{attribute 'GeneratedUsingTerminal: EP5001-0002-0016'}
{attribute addProperty BoxType "EP5001-0002-0016"}
{attribute addProperty Id "SSI_InputsAT %I*SSI_Inputs_0E3D8E3310WcStateAT %I*WcState_9091E0EB2InfoDataAT %I*InfoData_32EB74EA10"}
{attribute addProperty CRC "187224199"}
{attribute addProperty Size "22"}
TYPE EP5001_0B28D087 EXTENDS EtcSlaveTerminalBase_947E5A46 :
STRUCT
	{attribute addProperty Name "SSI_Inputs"}
	SSI_Inputs : SSI_Inputs_0E3D8E33;
	{attribute addProperty Name "WcState"}
	WcState : WcState_9091E0EB;
	{attribute addProperty Name "InfoData"}
	InfoData : InfoData_32EB74EA;
END_STRUCT
END_TYPE

(* stored: Version 1.2.0.0, ProductVersion 3.1.4024.9
   DUT EP5001_0B28D087: Id {dd714dfa-f178-4a90-9c10-4c57fcfea7b1} *)
